SUBAPPLICATION PublishEventHTTPPartial (* Publish Event using HTTP. The system and event information are encapsulated *)
  (* Standard: 61499-2; Description: Copyright (c) 2019 fortiss GmbH This program and the accompanying materials are made SPDX-License-Identifier: EPL-2.0 *)
  (* Version 1.0, 2019-11-12, Jose Cabral, fortiss GmbH *)
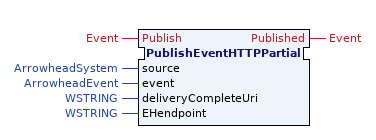
  EVENT_INPUT
    Publish;
  END_EVENT
  EVENT_OUTPUT
    Published;
  END_EVENT
  VAR_INPUT
    source : ArrowheadSystem; (* ArrowheadSystem publishing the event *)
    event : ArrowheadEvent; (* The published event *)
    deliveryCompleteUri : WSTRING; (* The URL subpath the Event Handler can use to inform the publisher about the results of the event propagation. If null, the Event Handler will not try to send the results *)
    EHendpoint : WSTRING; (* Endpoint (IP:PORT/URI) of the Event Handler (not officially in the documentation, but it simplifies the FBs) *)
  END_VAR
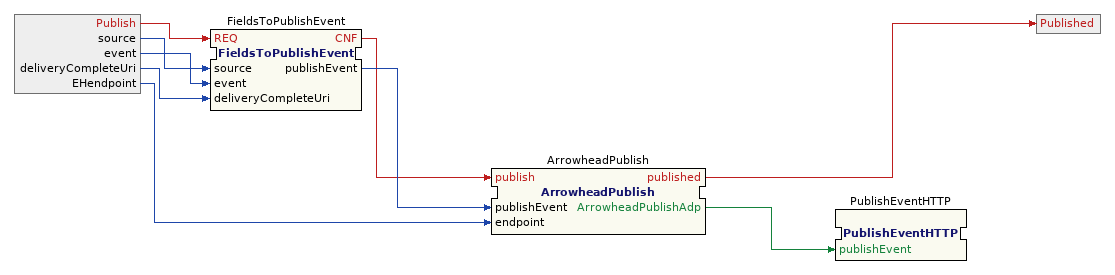
  FBS
    ArrowheadPublish : ArrowheadPublish;
    FieldsToPublishEvent : FieldsToPublishEvent;
    PublishEventHTTP : PublishEventHTTP;
  END_FBS
  EVENT_CONNECTIONS
    FieldsToPublishEvent.CNF TO ArrowheadPublish.publish;
    ArrowheadPublish.published TO Published;
    Publish TO FieldsToPublishEvent.REQ;
  END_CONNECTIONS
  DATA_CONNECTIONS
    FieldsToPublishEvent.publishEvent TO ArrowheadPublish.publishEvent;
    source TO FieldsToPublishEvent.source;
    event TO FieldsToPublishEvent.event;
    deliveryCompleteUri TO FieldsToPublishEvent.deliveryCompleteUri;
    EHendpoint TO ArrowheadPublish.endpoint;
  END_CONNECTIONS
  ADAPTER_CONNECTIONS
    ArrowheadPublish.ArrowheadPublishAdp TO PublishEventHTTP.publishEvent;
  END_CONNECTIONS
END_SUBAPPLICATION
